{attribute 'linkalways'}
{attribute 'hide_all_locals'}
FUNCTION_BLOCK ValueByte EXTENDS ValueByteRead IMPLEMENTS Value
VAR
END_VAR

METHOD SetFromType : BOOL
VAR_INPUT
	source : __SYSTEM.AnyType;
END_VAR
SetFromType := ConvertAnyType(source, thisAnyType);
END_METHOD

METHOD SetFromString : BOOL
VAR_INPUT
	value : T_MaxString;
END_VAR
thisValue := STRING_TO_BYTE(value);

SetFromString := TRUE;
END_METHOD

METHOD Set : BOOL
VAR_INPUT
	source : ANY;
END_VAR
Set := ConvertAnyType(source, thisAnyType);
END_METHOD

END_FUNCTION_BLOCK

(* stored: Version 1.1.0.1
   POU ValueByte: Id {33be5b33-c7e9-4cc4-ae2b-b1ca3d951fcd}, SpecialFunc None
   Method SetFromType: Id {027a1e04-5fd1-4381-91a2-99ad6bca9e51}
   Method SetFromString: Id {880f3e3d-fd25-4c42-bb3f-a135d686e515}
   Method Set: Id {d0fa0c61-cdd7-4766-bf96-0bb65b05174e} *)
